FUNCTION_BLOCK FB_Clock
(*
Square wave oscillator

Copyright (c) 2009-2017 victortorreslopez

GNU General Public License

Version history
2.1, 2017/03/15, VTL: style review (PLCopen Coding Guidelines)
2.0, 2014/12/29, VTL: complete review
1.0, 2009/11/06, VTL: first release
0.0, 2009/11/06, VTL: alfa release
*)
VAR_INPUT
  EN: BOOL := TRUE;	(* ENabled *)
  PT: TIME := T#500ms; (* Semicycle time *)
END_VAR
VAR_OUTPUT
  ET: TIME; (* Elapsed time *)
  Q: BOOL; (* Square wave *)
END_VAR
VAR
  Timer: TON; (* Auto-pilot timer *)
END_VAR

(* OUTPUT FUNCTION *)
IF Timer.Q THEN
  Q := NOT Q;
END_IF

(* FUNCTION BLOCKS *)
Timer(IN := EN AND NOT Timer.Q, PT := PT, ET => ET);

END_FUNCTION_BLOCK

(* stored: Version 1.1.0.1, ProductVersion 3.1.4024.12
   POU FB_Clock: Id {0fdf1c64-08a9-4609-bd01-9d0a87e1463c}, SpecialFunc None *)
